// PLC global variables
{attribute 'qualified_only'}
VAR_GLOBAL
    AMSNetId AT %I* : AMSNETID;
END_VAR

(* stored: Version 1.1.0.1, ProductVersion 3.1.4022.18
   GVL GVL_PLC: Id {427ac7fa-93f9-46f1-a3bb-0e3bcdb64033} *)
